(* IEC 61131-3 sources: windowtracking/src/Window, 7 files *)

(* ---- ITransportWindow.st ---- *)
USING Simatic.Ax.WindowTracking.Exits;
USING Simatic.Ax.SimpleControlModules;

NAMESPACE Simatic.Ax.WindowTracking
    INTERFACE ITransportWindow

        METHOD Reset
        END_METHOD

        METHOD CalcPosition : BOOL
            VAR_INPUT
                enc : IEncoder;
            END_VAR
        END_METHOD

        METHOD GetPosition : DINT
        END_METHOD

    END_INTERFACE
END_NAMESPACE

(* ---- ITransportWindowsCleanup.st ---- *)
USING Simatic.Ax.WindowTracking.Trigger;
USING Simatic.Ax.SimpleControlModules;

NAMESPACE Simatic.Ax.WindowTracking
    INTERFACE ITransportWindowsCleanup

        METHOD Remove
        END_METHOD

    END_INTERFACE
END_NAMESPACE

(* ---- ITransportWindowsTerminate.st ---- *)
NAMESPACE Simatic.Ax.WindowTracking
    INTERFACE ITransportWindowsTerminate

        METHOD Terminate
        END_METHOD

    END_INTERFACE
END_NAMESPACE

(* ---- ClearWindowTest.st ---- *)
USING AxUnit.Assert;
USING Simatic.Ax.WindowTracking.Events;
USING Simatic.Ax.WindowTracking.Trigger;

NAMESPACE Simatic.Ax.WindowTracking.EventHandler
    {TestFixture}
    CLASS ClearWindowTest
        VAR PROTECTED
            tws : TransportWindowList;
            enc : EncoderMock;
            v1 : VirtualTrigger := (Position := 100, Id := UINT#1);
            v2 : VirtualTrigger := (Position := 200, Id := UINT#2);
            te1 : TriggerEventMock;
            te2 : ClearWindow;
            tl : TriggerList;
        END_VAR

        METHOD PROTECTED Setup
            tws.Encoder := enc;
            v1.EventHandler := te1;
            v2.EventHandler := te2;
            te2.WindowList := tws;
            tl.Add(v1);
            tl.Add(v2);
            tws.TriggerPointList := tl;
        END_METHOD

        {Test}
        METHOD PUBLIC MyTestMethod
            THIS.Setup();
            tws.Create();
            enc.EncoderValue := 0;
            tws.Evaluate();
            Equal(expected := UINT#1, actual := tws.Count());

            enc.EncoderValue := 100;
            tws.Create();
            tws.Evaluate();
            Equal(expected := UINT#2, actual := tws.Count());

            // Remove Window at Position 200
            enc.EncoderValue := 200;
            tws.Evaluate();
            Equal(expected := UINT#1, actual := tws.Count());

        END_METHOD
    END_CLASS
END_NAMESPACE

(* ---- TransportWindow.st ---- *)
USING Simatic.Ax.SimpleControlModules;
USING Simatic.Ax.WindowTracking.Items;
NAMESPACE Simatic.Ax.WindowTracking

    CLASS TransportWindow IMPLEMENTS ITransportWindow
        VAR PUBLIC
            Item : IItem;
        END_VAR
        VAR PROTECTED
            _actualPos : DINT;
            _lastPos : DINT := -1;
        END_VAR

        METHOD PUBLIC CalcPosition : BOOL
            VAR_INPUT
                enc : IEncoder;
            END_VAR
            VAR_TEMP
                _newPos : DINT;
                _difference : DINT;
            END_VAR
            IF enc = NULL THEN
                CalcPosition := FALSE;
                RETURN;
            END_IF;
            IF (_lastPos = -1) THEN
                _lastPos := enc.GetValue();
            END_IF;
            _newPos := enc.GetValue();
            _difference := (_newPos - _lastPos + enc.GetModulo()) MOD enc.GetModulo();
            _actualPos := _actualPos + _difference;
            _lastPos := _newPos;
            CalcPosition := TRUE;
        END_METHOD

        METHOD PUBLIC GetPosition : DINT
            GetPosition := _actualPos;
        END_METHOD

        METHOD PUBLIC Reset
            _actualPos := 0;
            _lastPos := -1;
        END_METHOD

        METHOD PUBLIC GetItem : IItem
            GetItem := Item;
        END_METHOD
    END_CLASS
END_NAMESPACE

(* ---- TransportWindowList.st ---- *)
USING Simatic.Ax.WindowTracking.Trigger;
USING Simatic.Ax.SimpleControlModules;

NAMESPACE Simatic.Ax.WindowTracking
    CLASS TransportWindowList IMPLEMENTS ITransportWindowsCleanup
        VAR PUBLIC
            Encoder : IEncoder;
            TriggerPointList : ITriggerList;
        END_VAR
        VAR PROTECTED
            _tranportWindowList : ARRAY[UINT#0..BUF_SIZE - UINT#1] OF ITransportWindow;
            _tranportWindowListStorage : ARRAY[UINT#0..BUF_SIZE - UINT#1] OF TransportWindow;
            _count : UINT;
            _head : UINT;
            _tail : UINT;
        END_VAR

        VAR CONSTANT
            BUF_SIZE : UINT := UINT#100;
        END_VAR

        METHOD PUBLIC Create : ITransportWindow
            IF (Encoder = NULL) THEN
                Create := NULL;
                RETURN;
            END_IF;

            _tranportWindowList[_head] := _tranportWindowListStorage[_head];
            _tranportWindowList[_head].CalcPosition(Encoder);
            Create := _tranportWindowList[_head];

            _head := _head + UINT#1;
            _head := _head MOD BUF_SIZE;
        END_METHOD

        METHOD PUBLIC Remove
            IF (_tranportWindowList[_tail] <> NULL) THEN
                _tranportWindowListStorage[_tail].Reset();
                _tranportWindowList[_tail] := NULL;
                _tail := _tail + UINT#1;
                _tail := _tail MOD BUF_SIZE;
            END_IF;
        END_METHOD

        METHOD PUBLIC GetWindow : ITransportWindow
             VAR_INPUT
                 id : UINT;
             END_VAR
             GetWindow := _tranportWindowListStorage[id];
        END_METHOD

        METHOD PUBLIC Count : UINT
            Count := ((_head - _tail) + BUF_SIZE) MOD BUF_SIZE;
        END_METHOD

        METHOD PUBLIC Evaluate : BOOL
            VAR_TEMP
                i : UINT;
                o : ITransportWindow;
            END_VAR

            FOR i := UINT#0 TO THIS.Count() - UINT#1 DO
                o := _tranportWindowList[(_tail + i) MOD BUF_SIZE];
                IF (o <> NULL) THEN
                    o.CalcPosition(enc := Encoder);
                    IF (TriggerPointList <> NULL) THEN
                        TriggerPointList.Check(o);
                        Evaluate := TRUE;
                    ELSE
                        Evaluate := FALSE;
                    END_IF;
                END_IF;
            END_FOR;

        END_METHOD
    END_CLASS
END_NAMESPACE

(* ---- TransportWindows.st ---- *)
USING Simatic.Ax.WindowTracking.Trigger;
USING Simatic.Ax.SimpleControlModules;

NAMESPACE Simatic.Ax.WindowTracking
    CLASS TransportWindows
        VAR PUBLIC
            Encoder : IEncoder;
            TriggerPointList : ITriggerList;
        END_VAR
        VAR PROTECTED
            _tranportWindowList : ARRAY[UINT#0..BUF_SIZE - UINT#1] OF ITransportWindow;
            _tranportWindowListStorage : ARRAY[UINT#0..BUF_SIZE - UINT#1] OF TransportWindow;
            _count : UINT;
            _head : UINT;
            _tail : UINT;
        END_VAR

        VAR CONSTANT
            BUF_SIZE : UINT := UINT#100;
        END_VAR

        METHOD PUBLIC Create : ITransportWindow
            IF (Encoder = NULL) THEN
                Create := NULL;
                RETURN;
            END_IF;

            _tranportWindowList[_head] := _tranportWindowListStorage[_head];
            _tranportWindowList[_head].CalcPosition(Encoder);
            Create := _tranportWindowList[_head];

            _head := _head + UINT#1;
            _head := _head MOD BUF_SIZE;
        END_METHOD

        METHOD PUBLIC Remove
            IF (_tranportWindowList[_tail] <> NULL) THEN
                _tranportWindowListStorage[_tail].Reset();
                _tranportWindowList[_tail] := NULL;
                _tail := _tail + UINT#1;
                _tail := _tail MOD BUF_SIZE;
            END_IF;
        END_METHOD

        METHOD PUBLIC GetWindow : ITransportWindow
             VAR_INPUT
                 id : UINT;
             END_VAR
             GetWindow := _tranportWindowListStorage[id];
        END_METHOD

        METHOD PUBLIC Count : UINT
            Count := ((_head - _tail) + BUF_SIZE) MOD BUF_SIZE;
        END_METHOD

        METHOD PUBLIC Evaluate : BOOL
            VAR_TEMP
                i : UINT;
                o : ITransportWindow;
            END_VAR

            FOR i := UINT#0 TO THIS.Count() - UINT#1 DO
                o := _tranportWindowList[(_tail + i) MOD BUF_SIZE];
                IF (o <> NULL) THEN
                    o.CalcPosition(enc := Encoder);
                    IF (TriggerPointList <> NULL) THEN
                        TriggerPointList.Check(o);
                        Evaluate := TRUE;
                    ELSE
                        Evaluate := FALSE;
                    END_IF;
                END_IF;
            END_FOR;

        END_METHOD
    END_CLASS
END_NAMESPACE
